Staubli VAL3: setAllAccel.pgx

public program setAllAccel(num x_nNewValue, num x_nOldValue)
  local num i
  local num l_nSize
begin
end
